// TIA Portal V17 export
// export: Created 2021-12-03T08:13:13.6703667Z, ExportSetting WithDefaults, DisplayName Totally Integrated Automation Portal, DisplayVersion V17, DisplayName TIA Portal Openness, DisplayVersion V17, DisplayName TIA Portal Version Control Interface, DisplayVersion V17, DisplayName STEP 7 Professional, DisplayVersion V17, DisplayName STEP 7 Safety, DisplayVersion V17, DisplayName WinCC Advanced, DisplayVersion V17
DATA_BLOCK "FGDB_Simulation"   // DB80, F_DB
VERSION : 0.1
// stored: AutoNumber false
   VAR
      "/EmStpAccCon_Ch1" : Bool;   // Консоль ускорителя канал 1
      "/EmStpP1_Ch1" : Bool;   // Пульт Р1 канал 1
      "/EmStpP2_Ch1" : Bool;   // Пульт Р2 канал 1
      PrDoor1Cls_Ch1 : Bool;   // Замок блокирующий дверь 1 канал 1
      PrDoor2Cls_Ch1 : Bool;   // Замок блокирующий дверь 2 канал 1
      Spare40_5 : Bool;   // Spare
      "/EmStpDosimeter_Ch1" : Bool;   // Дозиметр канал 1
      PrDoor1Req : Bool;   // Запрос на открытие двери 1
      P3AckInSArea_Ch1 : Bool;   // Сброс внутри периметра безопасности
      FBPowerModulator : Bool;   // Обратная связь модулятора
      FBPowerConveyor : Bool;   // Обратная связь частотного преобразователя
      FBPowerXRayUnit : Bool;   // Обратная связь ускоритель
      "/EmStpAccCon_Ch2" : Bool;   // Консоль ускорителя канал 2
      "/EmStpP1_Ch2" : Bool;   // Пульт Р1 канал 2
      "/EmStpP2_Ch2" : Bool;   // Пульт Р2 канал 2
      PrDoor1Cls_Ch2 : Bool;   // Замок блокирующий дверь 1 канал 2
      PrDoor2Cls_Ch2 : Bool;   // Замок блокирующий дверь 2 канал 2
      Spare42_2 : Bool;   // Spare
      "/EmStpDosimeter_Ch2" : Bool;   // Дозиметр канал 2
      PrDoor2Req : Bool;   // Запрос на открытие двери 2
      P1AckEmStpOutSArea : Bool;   // Сброс снаружи периметра безопасности
      FBPowerChiller : Bool;   // Обратная связь чиллер
      FBPower_AccConsol : Bool;   // Обратная связь консоль ускорителя
      FBPowerModulator1P : Bool;   // Обратная связь модулятора 1 фаза
      "/EmStpP3_Ch1" : Bool;   // Пульт P3 канал 1
      P2AgreeBut_Ch1 : Bool;   // Кнопка разрешения канал 1
      Spare60_2 : Bool;   // Spare
      Spare60_3 : Bool;   // Spare
      Spare60_4 : Bool;   // Spare
      Spare60_5 : Bool;   // Spare
      Spare60_6 : Bool;   // Spare
      Spare60_7 : Bool;   // Spare
      P1KeyGenRel_Ch1 : Bool;   // Главный ключ разрешения канал 1
      P1KeyAccRel_Ch1 : Bool;   // Ключ разрешения включения ускорителя канал 1
      Spare61_2 : Bool;   // Spare
      Spare61_3 : Bool;   // Spare
      "/EmStpP3_Ch2" : Bool;   // Пульт P3 канал 2
      P2AgreeBut_Ch2 : Bool;   // Кнопка разрешения канал 2
      Spare61_6 : Bool;   // Spare
      Spare61_7 : Bool;   // Spare
      Spare62_0 : Bool;   // Spare
      Spare62_1 : Bool;   // Spare
      Spare62_2 : Bool;   // Spare
      Spare62_3 : Bool;   // Spare
      P1KeyGenRel_Ch2 : Bool;   // Главный ключ разрешения канал 2
      P1KeyAccRel_Ch2 : Bool;   // Ключ разрешения включения ускорителя канал 2
      Spare62_6 : Bool;   // Spare
      Spare62_7 : Bool;   // Spare
   END_VAR
BEGIN
END_DATA_BLOCK
